Universal Robots PolyScope program: Pick_n_Place1.urp

Program Pick_n_Place1 (createdIn=3.0.0 lastSavedIn=3.0.0 directory=/programs installation=default)
Robot Program (runOnlyOnce=true motionType=MoveJ speed=1.047198 acceleration=1.396263 useActiveTCP=false)
  'Program generated by RoboDK v5.3.2 for UR5e on 20/01/2022 14:09:03'
  'Using nominal kinematics.'
  Call approach_t1
  Call openGripper
  Call move_t1
  Call closeGripper
  Call deppr_t1
  Call approach_t2
  Call move_t2
  Call openGripper
  Call deppr_t2
  Call closeGripper
SubProgram -> approach_t1
SubProgram -> openGripper
SubProgram -> move_t1
SubProgram -> closeGripper
SubProgram -> deppr_t1
SubProgram -> approach_t2
SubProgram -> move_t2
SubProgram -> deppr_t2
SubProgram approach_t1 (keepSynchronizedWithDisk=true trackProgramExecution=false) programFile=/programs/approach_t1.urp
SubProgram openGripper (keepSynchronizedWithDisk=true trackProgramExecution=false) programFile=/programs/openGripper.urp
SubProgram move_t1 (keepSynchronizedWithDisk=true trackProgramExecution=false) programFile=/programs/move_t1.urp
SubProgram closeGripper (keepSynchronizedWithDisk=true trackProgramExecution=false) programFile=/programs/closeGripper.urp
SubProgram deppr_t1 (keepSynchronizedWithDisk=true trackProgramExecution=false) programFile=/programs/deppr_t1.urp
SubProgram approach_t2 (keepSynchronizedWithDisk=true trackProgramExecution=false) programFile=/programs/approach_t2.urp
SubProgram move_t2 (keepSynchronizedWithDisk=true trackProgramExecution=false) programFile=/programs/move_t2.urp
SubProgram deppr_t2 (keepSynchronizedWithDisk=true trackProgramExecution=false) programFile=/programs/deppr_t2.urp
